(* IEC 61131-3 sources: SMART-IRRIGATION-OPTIMIZATION-SYSTEM/milestone1, 1 file *)

(* ---- SmartIrrigation.st ---- *)
(*SmartIrrigation.st
 * ST (IEC 61131-3) Implementation for Smart Irrigation Optimization System
 * Milestone 1
*)

PROGRAM SmartIrrigation
  VAR
    status: STRING := 'Milestone 1';
  END_VAR

  (* Placeholder for Structured Text implementation *)
END_PROGRAM
